// TIA Portal V19 export
FUNCTION "Generic_CALL" : Void   // FC118, LAD
// stored: SetENOAutomatically false
BEGIN

REGION Network 2
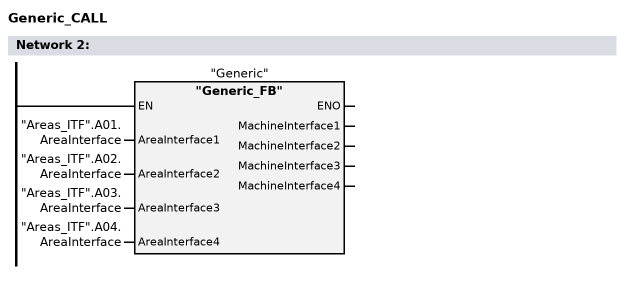
   RUNG wire#powerrail
      "Generic"(AreaInterface1 := "Areas_ITF".A01.AreaInterface, AreaInterface2 := "Areas_ITF".A02.AreaInterface, AreaInterface3 := "Areas_ITF".A03.AreaInterface, AreaInterface4 := "Areas_ITF".A04.AreaInterface, MachineInterface1 =>, MachineInterface2 =>, MachineInterface3 =>, MachineInterface4 =>)
   END_RUNG
   // the same network as SCL:
   "Generic"(AreaInterface1 := "Areas_ITF".A01.AreaInterface,   // "Generic_FB"
             AreaInterface2 := "Areas_ITF".A02.AreaInterface,
             AreaInterface3 := "Areas_ITF".A03.AreaInterface,
             AreaInterface4 := "Areas_ITF".A04.AreaInterface);
END_REGION
END_FUNCTION
